{attribute 'qualified_only'}
VAR_GLOBAL
	stMotor1 : ST_MotorParameters;
	stMotor2 : ST_MotorParameters;
END_VAR

(* stored: Version 1.1.0.1, ProductVersion 3.1.4024.12
   GVL GVL_Task3: Id {a99bf708-c3b3-430b-bf2e-730add40c24c} *)
